(* IEC 61131-3 sources: SRCI/RobotLibrary/RobotLibrary/Functions/Swap, 8 files *)

(* ---- GetHalfeByteHi.st ---- *)
FUNCTION GetHalfeByteHi : BYTE
VAR_INPUT
  /// Increase payload pointer
  Value : BYTE;
END_VAR

  GetHalfeByteHi.0 := Value.4;
  GetHalfeByteHi.1 := Value.5;
  GetHalfeByteHi.2 := Value.6;
  GetHalfeByteHi.3 := Value.7;

END_FUNCTION

(* ---- GetHalfeByteLo.st ---- *)
FUNCTION GetHalfeByteLo : BYTE
VAR_INPUT
  /// Increase payload pointer
  Value : BYTE;
END_VAR

  GetHalfeByteLo.0 := Value.0;
  GetHalfeByteLo.1 := Value.1;
  GetHalfeByteLo.2 := Value.2;
  GetHalfeByteLo.3 := Value.3;

END_FUNCTION

(* ---- SwapBytes.st ---- *)
FUNCTION SwapBytes
// -------------------------------------------------------------------------
//  SRCI Robot Library
// -------------------------------------------------------------------------
//
//  Object:      SwapBytes
//  Author:      Thorsten Brach
//  Date:        2024-06-01
//
//  Description:
//
//
//  Copyright:
//    (C) 2024 Thorsten Brach. All rights reserved
//             Licensed under the LGPL-3.0 license.
//
//  Disclaimer:
//    This project is provided without any guarantee and can be used for
//    private and commercial purposes. Any use is at the user’s
//    own risk and responsibility.
//
// -------------------------------------------------------------------------
VAR_INPUT
  /// pointer to data type
  pValue : POINTER TO BYTE;
  /// size of data type
  Size  : UDINT;
END_VAR

VAR
  /// Pointer to low word low byte
  _pLwLb    : POINTER TO BYTE;
  /// Pointer to low word high byte
  _pLwHb    : POINTER TO BYTE;
  /// Pointer to high word low byte
  _pHwLb    : POINTER TO BYTE;
  /// Pointer to high word high byte
  _pHwHb    : POINTER TO BYTE;
   /// temporary bytes
  _tmpBytes : ARRAY[1..4] OF BYTE;
END_VAR

  IF ( RobotLibraryParameter.SWAP_BYTE_ORDER AND Size = 2)
  THEN
   _pLwLb := pValue + 0;
   _pLwHb := pValue + 1;

    // swap bytes
   _tmpBytes[1] := _pLwHb^;
   _tmpBytes[2] := _pLwLb^;

    // copy bytes to data type
    MemCpy(pValue, ADR(_tmpBytes), Size);
  END_IF

  IF ( RobotLibraryParameter.SWAP_BYTE_ORDER AND Size = 4)
  THEN
   _pLwLb := pValue + 0;
   _pLwHb := pValue + 1;
   _pHwLb := pValue + 2;
   _pHwHb := pValue + 3;

    // swap bytes
   _tmpBytes[1] := _pHwHb^;
   _tmpBytes[2] := _pHwLb^;
   _tmpBytes[3] := _pLwHb^;
   _tmpBytes[4] := _pLwLb^;

    // copy bytes to data type
    MemCpy(pValue, ADR(_tmpBytes),Size);
  END_IF

END_FUNCTION

(* ---- SwapDword.st ---- *)
FUNCTION SwapDword : DWORD
// -------------------------------------------------------------------------
//  SRCI Robot Library
// -------------------------------------------------------------------------
//
//  Object:      SwapDword
//  Author:      Thorsten Brach
//  Date:        2024-06-01
//
//  Description:
//
//
//  Copyright:
//    (C) 2024 Thorsten Brach. All rights reserved
//             Licensed under the LGPL-3.0 license.
//
//  Disclaimer:
//    This project is provided without any guarantee and can be used for
//    private and commercial purposes. Any use is at the user’s
//    own risk and responsibility.
//
// -------------------------------------------------------------------------
VAR_INPUT
  /// Value
  Value : DWORD;
END_VAR

  SwapBytes(ADR(Value),SIZEOF(Value));

  SwapDword := Value;

END_FUNCTION

(* ---- SwapIecDate.st ---- *)
FUNCTION SwapIecDate : IEC_DATE
// -------------------------------------------------------------------------
//  SRCI Robot Library
// -------------------------------------------------------------------------
//
//  Object:      SwapIecDate
//  Author:      Thorsten Brach
//  Date:        2024-06-09
//
//  Description:
//
//
//  Copyright:
//    (C) 2024 Thorsten Brach. All rights reserved
//             Licensed under the LGPL-3.0 license.
//
//  Disclaimer:
//    This project is provided without any guarantee and can be used for
//    private and commercial purposes. Any use is at the user’s
//    own risk and responsibility.
//
// -------------------------------------------------------------------------
VAR_INPUT
  /// Value to swap
  Value : IEC_DATE;
END_VAR

  SwapBytes(ADR(Value),SIZEOF(Value));

  SwapIecDate := Value;

END_FUNCTION

(* ---- SwapIecTime.st ---- *)
FUNCTION SwapIecTime : TOD
// -------------------------------------------------------------------------
//  SRCI Robot Library
// -------------------------------------------------------------------------
//
//  Object:      SwapTime
//  Author:      Thorsten Brach
//  Date:        2024-06-01
//
//  Description:
//
//
//  Copyright:
//    (C) 2024 Thorsten Brach. All rights reserved
//             Licensed under the LGPL-3.0 license.
//
//  Disclaimer:
//    This project is provided without any guarantee and can be used for
//    private and commercial purposes. Any use is at the user’s
//    own risk and responsibility.
//
// -------------------------------------------------------------------------
VAR_INPUT
  /// Value
  Value : TOD;
END_VAR

  SwapBytes(ADR(Value),SIZEOF(Value));

  SwapIecTime := Value;

END_FUNCTION

(* ---- SwapInt.st ---- *)
FUNCTION SwapInt : INT
// -------------------------------------------------------------------------
//  SRCI Robot Library
// -------------------------------------------------------------------------
//
//  Object:      SwapInt
//  Author:      Thorsten Brach
//  Date:        2024-06-01
//
//  Description:
//
//
//  Copyright:
//    (C) 2024 Thorsten Brach. All rights reserved
//             Licensed under the LGPL-3.0 license.
//
//  Disclaimer:
//    This project is provided without any guarantee and can be used for
//    private and commercial purposes. Any use is at the user’s
//    own risk and responsibility.
//
// -------------------------------------------------------------------------
VAR_INPUT
  /// Value to swap
  Value : INT;
END_VAR

  SwapBytes(ADR(Value),SIZEOF(Value));

  SwapInt := Value;

END_FUNCTION

(* ---- SwapWord.st ---- *)
FUNCTION SwapWord : WORD
// -------------------------------------------------------------------------
//  SRCI Robot Library
// -------------------------------------------------------------------------
//
//  Object:      SwapWord
//  Author:      Thorsten Brach
//  Date:        2024-06-01
//
//  Description:
//
//
//  Copyright:
//    (C) 2024 Thorsten Brach. All rights reserved
//             Licensed under the LGPL-3.0 license.
//
//  Disclaimer:
//    This project is provided without any guarantee and can be used for
//    private and commercial purposes. Any use is at the user’s
//    own risk and responsibility.
//
// -------------------------------------------------------------------------
VAR_INPUT
  /// Value to swap
  Value : UINT;
END_VAR

  SwapBytes(ADR(Value),SIZEOF(Value));

  SwapWord := Value;

END_FUNCTION
